{attribute 'qualified_only'}
TYPE E_MMDirection :
(
	eMMDirection_BiDirectional	:= 0,																				(**)
	eMMDirection_Forward		:= 1,																				(**)
	eMMDirection_Backward		:= 2																				(**)
) BYTE;
END_TYPE

(* stored: Version 1.1.0.1, ProductVersion 3.1.4024.5
   EnumerationTextList E_MMDirection: Id {44b8e322-6dea-49ad-854e-bda197468b3c} *)
